// Packed ARGB color value.
TYPE Argb : DWORD; END_TYPE

(* stored: Version 1.1.0.1
   DUT Argb: Id {ac8fa48f-31f7-4a96-8768-9b14bebd683c} *)
